{attribute 'GeneratedUsingTerminal: EP2328-1061-0016'}
{attribute addProperty BoxType "EP2328-1061-0016"}
{attribute addProperty Id "OutputAT %Q*BOOL1"}
{attribute addProperty CRC "1120571895"}
{attribute addProperty Size "1"}
TYPE DO_X04_Pin2_Output_42CA91F7 :
STRUCT
	{attribute addProperty Name "Output"}
	Output AT %Q* : BOOL;
END_STRUCT
END_TYPE

(* stored: Version 1.2.0.0, ProductVersion 3.1.4024.9
   DUT DO_X04_Pin2_Output_42CA91F7: Id {a21c79d0-feae-40d4-a867-e145f6a98104} *)
